FUNCTION_BLOCK FB_1stOrderFilter
VAR_INPUT
	bReset			: BOOL; (*Reset 1st order filter*)
	fIn				: REAL;	(*Input value*)
	fTime_1stFilter	: REAL;	(*First order filter time in seconds*)
	tTaskCycleTime	: TIME;

	//FB_CTRL_PT1: FB_CTRL_PT1;
END_VAR
VAR_OUTPUT
	fOut			: REAL; (*Output value 2nd Order filtered*)
END_VAR
VAR_IN_OUT

END_VAR

VAR
	bHold						: BOOL;
	bSync						: BOOL;
	bFilterActive				: BOOL;

	eMode						: E_CTRL_MODE;
	eState						: E_CTRL_STATE;

	FB_CTRL_PT1					: FB_CTRL_PT1;
	stCTRL_PT1_PARAMS			: ST_CTRL_PT1_PARAMS;
END_VAR

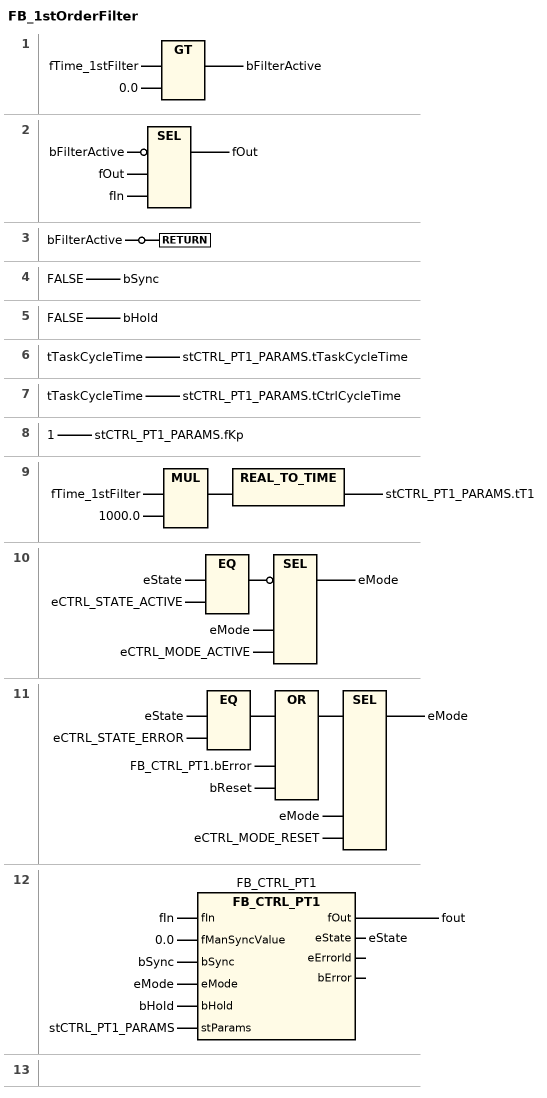
// NETWORK 1
bFilterActive := fTime_1stFilter > 0.0;

// NETWORK 2
fOut := SEL(NOT bFilterActive, fOut, fIn);

// NETWORK 3
IF NOT bFilterActive THEN RETURN; END_IF

// NETWORK 4
bSync := FALSE;

// NETWORK 5
bHold := FALSE;

// NETWORK 6
stCTRL_PT1_PARAMS.tTaskCycleTime := tTaskCycleTime;

// NETWORK 7
stCTRL_PT1_PARAMS.tCtrlCycleTime := tTaskCycleTime;

// NETWORK 8
stCTRL_PT1_PARAMS.fKp := 1;

// NETWORK 9
stCTRL_PT1_PARAMS.tT1 := REAL_TO_TIME(fTime_1stFilter * 1000.0);

// NETWORK 10
eMode := SEL(NOT (eState = eCTRL_STATE_ACTIVE), eMode, eCTRL_MODE_ACTIVE);

// NETWORK 11
eMode := SEL(eState = eCTRL_STATE_ERROR OR FB_CTRL_PT1.bError OR bReset, eMode, eCTRL_MODE_RESET);

// NETWORK 12
FB_CTRL_PT1(
    fIn := fIn,
    fManSyncValue := 0.0,
    bSync := bSync,
    eMode := eMode,
    bHold := bHold,
    stParams := stCTRL_PT1_PARAMS,
    eState => eState);
fout := FB_CTRL_PT1.fOut;

// NETWORK 13

END_FUNCTION_BLOCK

(* stored: Version 1.1.0.1, ProductVersion 3.1.4020.12
   POU FB_1stOrderFilter: Id {008e003a-cf6d-4332-ac72-cddf2969c672}, SpecialFunc None *)
